Fanuc KAREL source: shapes.kl

PROGRAM shapes
%NOBUSYLAMP
%COMMENT = 'shape functions'
%NOLOCKGROUP
%NOPAUSE = COMMAND + TPENABLE + ERROR

%include systemvars.klt
%include shapes.klt

%include math.klh
%include pose.klh
%include shapes.klh
%from systemlib.klh %import VEC, VEC2D

BEGIN
END shapes


ROUTINE shapes__create_plane
  BEGIN
    -- equation of plane ax+by+cz+d=0
    out_plane.origin = origin

    out_plane.normal = normal_vec/math__norm(normal_vec)
    -- solve for d
    out_plane.d = -1*(out_plane.normal@origin)
  END shapes__create_plane

ROUTINE shapes__create_plane_from_points
  VAR
    v1 : VECTOR
    v2 : VECTOR
    out_plane : t_PLANE
  BEGIN
    v1 = p2 - p1
    v2 = p3 - p1

    out_plane.normal = v1#v2
    out_plane.origin = p1
    out_plane.d = -1*(out_plane.normal@p1)

    RETURN(out_plane)
  END shapes__create_plane_from_points

ROUTINE shapes__project_point_on_plane
  BEGIN
    -- calculate distance from point to the plane
    -- move point back this distance along plane normal
    -- interect_point = P - D*n

    RETURN(point - shapes__distance_of_point_to_plane(point, plane) * plane.normal)
  END shapes__project_point_on_plane

ROUTINE shapes__distance_of_point_to_plane
  BEGIN
    -- calculate distance from point to the plane
    RETURN(plane.normal@point + plane.d)
  END shapes__distance_of_point_to_plane
